// Gets the upper bound index of the array of specified type.
FUNCTION F_GetTimeOfDayArrayUpperBound : T_Position // The upper bound index of the specified array.
VAR_IN_OUT
	arArray : ARRAY[*] OF TIME_OF_DAY; // The array to query.
END_VAR

F_GetTimeOfDayArrayUpperBound := UPPER_BOUND(arArray, 1);

END_FUNCTION

(* stored: Version 1.1.0.1
   POU F_GetTimeOfDayArrayUpperBound: Id {bfb9747e-6a6f-055d-032a-ce6ff804875e}, SpecialFunc None *)
